INTERFACE ITF_TopElement_HMI_Init EXTENDS ITF_TopElement, ITF_TopElement_HMI_Connector

END_INTERFACE

(* stored: Version 1.1.0.1, ProductVersion 3.1.4024.15
   Itf ITF_TopElement_HMI_Init: Id {a5a1df98-1b1f-4475-b4e2-808a736045a4} *)
